# EPICS StreamDevice protocol: ESP32_GPIO/protocols/ESP32_GPIO.protocol
Terminator = CR LF;

getDI
{
	out "DGET \$1";
	in "%{0|1}";
}
setDO
{
	out "DSET \$1 %i";
	in "OK";
	@init
	{out "DSET \$1 0";
	in "OK";}
}

getAI
{
	out "AGET \$1";
	in "%i";
}

setAO
{
	out "ASET \$1 %i";
	in "OK";
	@init
	{out "ASET \$1 0";
	in "OK";}
}

initDIO
{
	out "INIT \$1 \$2";
	in "OK";
}
